// TIA Portal V17 export
// export: Created 2025-03-05T08:01:07.6506648Z, ExportSetting WithDefaults, DisplayName Totally Integrated Automation Portal, DisplayVersion V17 Update 8, DisplayName TIA Portal Openness, DisplayVersion V17 Update 8, DisplayName TIA Portal Version Control Interface, DisplayVersion V17, DisplayName SINAMICS Startdrive Advanced, DisplayVersion V17 SP2, DisplayName SINAMICS Startdrive G110M, G120, G120C, G120D, G120P, G115D, DisplayVersion V17 SP2, DisplayName SINAMICS Startdrive G130, G150, S120, S150, SINAMICS MV, S210, DisplayVersion V17 SP2, DisplayName STEP 7 Professional, DisplayVersion V17 Update 8, DisplayName SINUMERIK ONE STEP 7 Toolbox, DisplayVersion V17 Update 12, DisplayName SINUMERIK 840D sl STEP 7 Toolbox, DisplayVersion V17 Update 12, DisplayName STEP 7 Safety, DisplayVersion V17 Update 6, DisplayName WinCC Advanced, DisplayVersion V17 Update 8
DATA_BLOCK "DB1013_SAFETY_CLADDING"   // DB1013, F_DB
{ DB_Accessible_From_OPC_UA := 'FALSE' }
AUTHOR : ETXETAR
VERSION : 1.0
// stored: AutoNumber false, DBAccessibleFromOPCUA false, DBAccessibleFromWebserver true, InstanceOfName FB1013_SAFETY_CLADDING, InstanceOfType FB
"FB1013_SAFETY_CLADDING"
   // VAR
   //    F_IEC_Timer_PWR_EN_DEL_2 : TOF;
   //    F_IEC_Timer_PWR_EN_DEL_3 : TOF;
   //    F_IEC_Timer_PWR_EN_DEL_4 : TOF;
   //    F_IEC_Timer_PWR_EN_RES_DEL : TON;
   //    F_IEC_Timer_PWR_EN_FDBCK : TON;
   //    F_IEC_Timer_GNTR_DR_FDBCK : TON;
   //    F_IEC_Timer_FIXT_WRK_COND_FDBCK : TON;
   //    F_IEC_Timer_MACHINE_E_STOP : TON;
   //    F_IEC_Timer_CLNT_OFF_01R : TOF;
   //    F_IEC_Timer_CLNT_OFF_01L : TOF;
   //    F_IEC_Timer_BIMANUAL_CLOSE : TON;
   // END_VAR
BEGIN
END_DATA_BLOCK
